PROGRAM PRG_UpdateFlowRateSensor
VAR
	deltaVolume : REAL := 0.0;
END_VAR

IF flowRateRawCounts < 20 THEN
	flowRateLitersPerMinute := 0.0;
ELSE
	flowRateLitersPerMinute := INT_TO_REAL(flowRateRawCounts)*flowRateCalibration.scaleFactor + flowRateCalibration.offset;
END_IF

deltaVolume := flowRateLitersPerMinute*0.01/60.0;
spargeVolume := spargeVolume + deltaVolume;
spargeVolumeCumulative := spargeVolumeCumulative+ deltaVolume;

IF  resetSpargeVolume THEN
	resetSpargeVolume := FALSE;
	spargeVolume := 0.0;
END_IF

IF resetSpargeVolumeCumulative THEN
	resetSpargeVolumeCumulative := FALSE;
	spargeVolumeCumulative := 0.0;
END_IF

END_PROGRAM

(* stored: Version 1.1.0.1, ProductVersion 3.1.4022.7
   POU PRG_UpdateFlowRateSensor: Id {98b19980-0f3a-4ba8-ae06-17189f6622e4}, SpecialFunc None *)
